FUNCTION_BLOCK Weight_cese
VAR_INPUT
	//W_Send :ST_Send;
	
END_VAR
VAR_IN_OUT

	W_Send :ST_SendData;
	W_Receive:ST_ReceiveData;
	W_Gross	:ST_Gross;
END_VAR
VAR_OUTPUT
	
	
END_VAR
VAR
	Step_W_Date :UINT;
	W_TON :ARRAY[1..6] OF Tc2_Standard.TON;
	strBetryName	:STRING;//字符串
	strBetryName2 	:STRING;
	strBetryName3 	:STRING;
	L_R: UDINT;
	L_S: UDINT;
	G_OUT1 	:STRING;
	G_OUT2 	:STRING;
	weight	:REAL;
	weight_Z	:REAL;
	WeightTestAgain :BOOL;
	WeightTestAgainMount :INT;
END_VAR

ACT();
W_TON[1](PT:=T#2S);
W_TON[2](PT:=T#100MS);
W_TON[3](PT:=T#2S);
W_TON[4](PT:=T#100MS);


//初始位称重功能块
IF W_Gross.Init THEN
	Step_W_Date:=0;
	W_Gross.Weight_start:=FALSE;
	W_Gross.Clear_start:=FALSE;
	W_Send.Status.InitRequest:=FALSE;
	W_Send.Status.TransmitRequest:=FALSE;
	W_Gross.error[1]:=FALSE;
	W_Gross.Clear_finish:=FALSE;
	W_Gross.Weight_finish:=FALSE;
	W_Gross.Init:=FALSE;
END_IF





CASE Step_W_Date  OF	
0://称重测试开始
IF W_Gross.Weight_start THEN
	Step_W_Date:=10;
	W_Gross.Weight_finish:=FALSE;
	W_Gross.Weight_start :=FALSE;
	W_Gross.Clear_finish:=FALSE;

ELSIF W_Gross.Clear_start THEN
	Step_W_Date:=1010;
	W_Gross.Clear_finish:=FALSE;
	W_Gross.Clear_start :=FALSE;
	W_Gross.Weight_finish:=FALSE;
END_IF

10://初始化
W_Send.Status.InitRequest:=TRUE;
W_TON[1].IN:=TRUE;
Step_W_Date:=20;

20://如果接收到就
IF W_Receive.Status.InitAccepted THEN
	Step_W_Date:=30;
	W_Send.Status.InitRequest:=FALSE;
	W_TON[1].IN:=FALSE;
END_IF
IF W_TON[1].Q THEN
	W_Send.Status.InitRequest:=FALSE;
	W_Gross.error[1]:=TRUE;
	W_TON[1].IN:=FALSE;
	Step_W_Date:=1111;
END_IF

30:
strBetryName:='Q$R$N';
STRING_TO_UTF8(pDstUTF8:=ADR(W_Send.Data) , pSrcSTRING:=ADR(strBetryName) , nDstSize:=INT_TO_UINT( LEN(STR:=strBetryName )+1));
W_Send.Status.OutputLength:=INT_TO_UINT( LEN(STR:=strBetryName ));
Step_W_Date:=40;

40:
W_Send.Status.TransmitRequest:=TRUE;
IF W_Receive.Status.TransmitDone AND W_Receive.Status.ReceiveRequest AND W_Receive.Status.TotalInputLength>5 THEN
	Step_W_Date:=50;
W_Send.Status.TransmitRequest:=FALSE;
END_IF

50:
L_R:=INT_TO_UDINT( LEN(STR:=strBetryName2 )+1);
UTF8_TO_STRING(pDstSTRING:=ADR(strBetryName2) , pSrcUTF8:=ADR(W_Receive.Data) , nDstSize:=SIZEOF(W_Receive.Data) , nDstLen=> L_R  );
W_TON[2].IN:=TRUE;
IF W_TON[2].Q THEN
Step_W_Date:=60;
W_TON[2].IN:=FALSE;
END_IF

60:
weight_Z:=STRING_TO_REAL(G_OUT2);
IF G_OUT1='+' THEN
	W_Gross.bweight:=weight_Z;
	Step_W_Date:=70;
END_IF
IF G_OUT1='-' THEN
	W_Gross.bweight:=-weight_Z;
	Step_W_Date:=70;
END_IF

70:
IF W_Gross.bweight >=1 OR WeightTestAgain THEN
W_Gross.Weight_finish:=TRUE;
Step_W_Date:=0;
WeightTestAgain:=FALSE;
ELSE
WeightTestAgain:=TRUE;
Step_W_Date:=10;
WeightTestAgainMount:=WeightTestAgainMount+1;
END_IF




1010://初始化
W_Send.Status.InitRequest:=TRUE;
W_TON[3].IN:=TRUE;
Step_W_Date:=1020;

1020://如果接收到就
IF W_Receive.Status.InitAccepted THEN
	Step_W_Date:=1030;
	W_Send.Status.InitRequest:=FALSE;
	W_TON[3].IN:=FALSE;
END_IF
IF W_TON[3].Q THEN
	W_Send.Status.InitRequest:=FALSE;
	W_Gross.error[1]:=TRUE;
	W_TON[3].IN:=FALSE;
	Step_W_Date:=1111;
END_IF

1030:
strBetryName3:='R$R$N';
STRING_TO_UTF8(pDstUTF8:=ADR(W_Send.Data) , pSrcSTRING:=ADR(strBetryName3) , nDstSize:=INT_TO_UINT( LEN(STR:=strBetryName3 )+1   )       );
W_Send.Status.OutputLength:=INT_TO_UINT( LEN(STR:=strBetryName3 ));
Step_W_Date:=1040;

1040:
W_Send.Status.TransmitRequest:=TRUE;
IF W_Receive.Status.TransmitDone  AND W_Receive.Status.ReceiveRequest THEN
	W_Send.Status.TransmitRequest:=FALSE;
	W_Send.Status.ReceiveAccepted:=TRUE;
	Step_W_Date:=1050;
END_IF

1050:
IF NOT W_Receive.Status.ReceiveRequest  THEN
	W_Send.Status.ReceiveAccepted:=FALSE;
	Step_W_Date:=1060;
END_IF

1060:
IF  W_Receive.Status.ReceiveRequest THEN
	W_Gross.Clear_finish:=TRUE;
	Step_W_Date:=0;
END_IF



END_CASE

ACTION ACT:
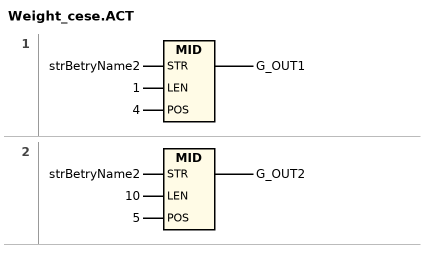
// NETWORK 1
G_OUT1 := MID(STR := strBetryName2, LEN := 1, POS := 4);

// NETWORK 2
G_OUT2 := MID(STR := strBetryName2, LEN := 10, POS := 5);
END_ACTION

END_FUNCTION_BLOCK

(* stored: Version 1.1.0.1, ProductVersion 3.1.4024.12
   POU Weight_cese: Id {4d0e4fbc-8712-477d-a6d6-d3283db8b9c1}, SpecialFunc None
   Action ACT: Id {4d624951-ef20-49f8-b78c-99228b9b80d0} *)
